// TIA Portal V15.1 export
// export: Created 2020-06-12T07:35:56.1474609Z, ExportSetting None, DisplayName Totally Integrated Automation Portal, DisplayVersion V15.1, DisplayName TIA Portal Openness, DisplayVersion V15.1, DisplayName STEP 7 Professional, DisplayVersion V15.1, DisplayName STEP 7 Safety, DisplayVersion V15.1, DisplayName WinCC Advanced, DisplayVersion V15.1
FUNCTION "MainSim" : Void   // FC193, FBD
{ S7_Optimized_Access := 'TRUE' }
// stored: SetENOAutomatically False
   VAR_TEMP
      tLso : Bool;
      tLsc : Bool;
      tTimeOut : Time;
      tPos : Real;
      tEncPID : DInt;
      tEncSensivity : LReal;
   END_VAR
BEGIN

REGION Network 1
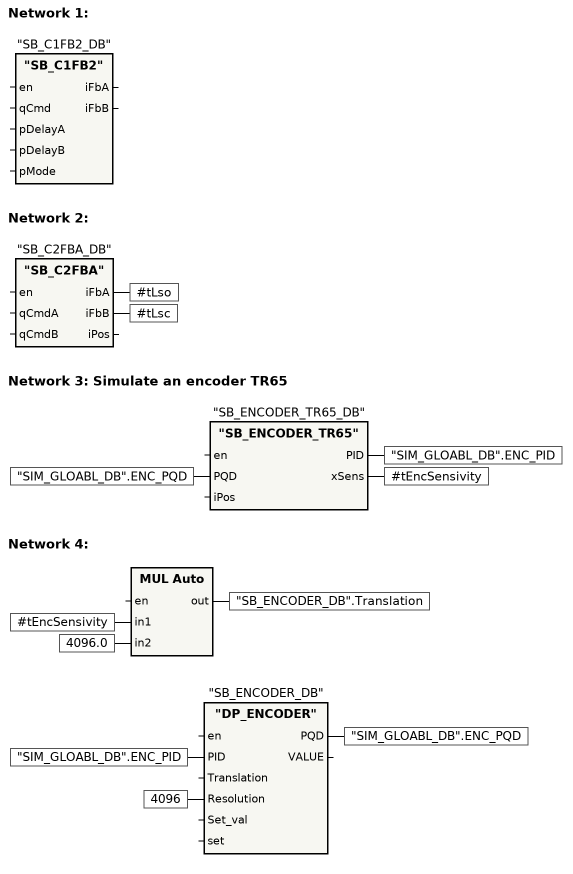
   "SB_C1FB2_DB"();   // "SB_C1FB2"
END_REGION

REGION Network 2
   "SB_C2FBA_DB"(iFbA => #tLso, iFbB => #tLsc);   // "SB_C2FBA"
END_REGION

REGION Network 3: Simulate an encoder TR65
   "SB_ENCODER_TR65_DB"(PQD := "SIM_GLOABL_DB".ENC_PQD, PID => "SIM_GLOABL_DB".ENC_PID, xSens => #tEncSensivity);   // "SB_ENCODER_TR65"
END_REGION

REGION Network 4
   "SB_ENCODER_DB".Translation := #tEncSensivity * 4096.0;
   "SB_ENCODER_DB"(PID := "SIM_GLOABL_DB".ENC_PID, Resolution := 4096, PQD => "SIM_GLOABL_DB".ENC_PQD);   // "DP_ENCODER"
END_REGION
END_FUNCTION
